(*

.. <legal notes>

legal notes
=================
| SPDX-FileCopyrightText: © 2026 Oleksandr Tiutyk <trofimich@gmail.com>
| SPDX-License-Identifier: LGPL-3.0-only
| For details check: LGPL-3.0-only_

.. _LGPL-3.0-only: https://www.gnu.org/licenses/lgpl-3.0.en.html

.. </legal notes>

*)

PROGRAM UsignedInt64Helper
VAR CONSTANT
	MIN_VALUE : ULINT := 0;
	MAX_VALUE : ULINT := 18_446_744_073_709_551_615;
END_VAR
VAR
	_ClassName : STRING := __POUNAME();
END_VAR

{attribute 'monitoring' := 'call'}
PROPERTY ClassName : STRING
GET
ClassName := _ClassName;
END_GET
END_PROPERTY

{attribute 'monitoring' := 'call'}
PROPERTY NamespaceName : STRING
GET
NamespaceName := CurrentNamespace.Name;
END_GET
END_PROPERTY

END_PROGRAM

(* stored: Version 1.1.0.1
   POU UsignedInt64Helper: Id {58df88cf-50aa-4336-8cc5-101184ba5ae9}, SpecialFunc None
   Property ClassName: Id {c9902b8b-4441-4db4-9836-61de8230deed}
   Get Get: Id {72636f1c-39cf-4e74-8ad7-9656e317c009}
   Property NamespaceName: Id {83f4fb94-795a-4980-a2a3-17badd4fcbbb}
   Get Get: Id {b608a452-9359-4c01-bfd0-24267a1c3c3b} *)
